{attribute 'GeneratedUsingTerminal: EK1100-0000-0018'}
{attribute addProperty BoxType "EK1100-0000-0018"}
{attribute addProperty Id "Beckhoff_EJ3xxxEK1122Beckhoff_EJ3xxxEK1122_F46733132A_0001_EJ3004_0000_0019EJ3004_9DDA7BAE48A_0002_EJ3004_0000_0020EJ3004_9DDA7BAE48A_0003_EJ3004_0000_0021EJ3004_9DDA7BAE48A_0004_EJ3048_0000_0020EJ3048_085DE50284A_0005_EJ3058_0000_0020EJ3058_085DE50284A_0006_EJ3068_0000_0020EJ3068_085DE50284A_0007_EJ3068_0000_0021EJ3068_085DE50284A_0008_EJ3104_0000_0019EJ3104_0E4717A052A_0009_EJ3104_0000_0020EJ3104_0E4717A052A_0010_EJ3104_0000_0021EJ3104_0E4717A052A_0011_EJ3108_0000_0017EJ3108_085DE50284A_0012_EJ3108_0000_0018EJ3108_5798389192A_0013_EJ3108_0000_0019EJ3108_5798389192A_0014_EJ3202_0000_0019EJ3202_14BDD8A530A_0015_EJ3202_0000_0020EJ3202_14BDD8A530A_0016_EJ3202_0000_0021EJ3202_14BDD8A530A_0017_EJ3214_0000_0016EJ3214_AFE9644F40A_0018_EJ3255_0000_0023EJ3255_6B0AD73762A_0019_EJ3318_0000_0017EJ3318_CF36AC5082"}
{attribute addProperty CRC "449149787"}
{attribute addProperty Size "1180"}
TYPE Beckhoff_EJ3xxx_1AC57B5B EXTENDS EK1100_AB5A9467 :
STRUCT
	{attribute addProperty Name "Beckhoff_EJ3xxxEK1122"}
	{attribute addProperty PreviousPort "Beckhoff EJ3xxx : B"}
	Beckhoff_EJ3xxxEK1122 : Beckhoff_EJ3xxxEK1122_F4673313;
	{attribute addProperty Name "A_0001_EJ3004_0000_0019"}
	{attribute addProperty PreviousPort "Beckhoff EJ3xxxEK1122 : C"}
	A_0001_EJ3004_0000_0019 : EJ3004_9DDA7BAE;
	{attribute addProperty Name "A_0002_EJ3004_0000_0020"}
	{attribute addProperty PreviousPort "A_0001(EJ3004-0000-0019) : B"}
	A_0002_EJ3004_0000_0020 : EJ3004_9DDA7BAE;
	{attribute addProperty Name "A_0003_EJ3004_0000_0021"}
	{attribute addProperty PreviousPort "A_0002(EJ3004-0000-0020) : B"}
	A_0003_EJ3004_0000_0021 : EJ3004_9DDA7BAE;
	{attribute addProperty Name "A_0004_EJ3048_0000_0020"}
	{attribute addProperty PreviousPort "A_0003(EJ3004-0000-0021) : B"}
	A_0004_EJ3048_0000_0020 : EJ3048_085DE502;
	{attribute addProperty Name "A_0005_EJ3058_0000_0020"}
	{attribute addProperty PreviousPort "A_0004(EJ3048-0000-0020) : B"}
	A_0005_EJ3058_0000_0020 : EJ3058_085DE502;
	{attribute addProperty Name "A_0006_EJ3068_0000_0020"}
	{attribute addProperty PreviousPort "A_0005(EJ3058-0000-0020) : B"}
	A_0006_EJ3068_0000_0020 : EJ3068_085DE502;
	{attribute addProperty Name "A_0007_EJ3068_0000_0021"}
	{attribute addProperty PreviousPort "A_0006(EJ3068-0000-0020) : B"}
	A_0007_EJ3068_0000_0021 : EJ3068_085DE502;
	{attribute addProperty Name "A_0008_EJ3104_0000_0019"}
	{attribute addProperty PreviousPort "A_0007(EJ3068-0000-0021) : B"}
	A_0008_EJ3104_0000_0019 : EJ3104_0E4717A0;
	{attribute addProperty Name "A_0009_EJ3104_0000_0020"}
	{attribute addProperty PreviousPort "A_0008(EJ3104-0000-0019) : B"}
	A_0009_EJ3104_0000_0020 : EJ3104_0E4717A0;
	{attribute addProperty Name "A_0010_EJ3104_0000_0021"}
	{attribute addProperty PreviousPort "A_0009(EJ3104-0000-0020) : B"}
	A_0010_EJ3104_0000_0021 : EJ3104_0E4717A0;
	{attribute addProperty Name "A_0011_EJ3108_0000_0017"}
	{attribute addProperty PreviousPort "A_0010(EJ3104-0000-0021) : B"}
	A_0011_EJ3108_0000_0017 : EJ3108_085DE502;
	{attribute addProperty Name "A_0012_EJ3108_0000_0018"}
	{attribute addProperty PreviousPort "A_0011(EJ3108-0000-0017) : B"}
	A_0012_EJ3108_0000_0018 : EJ3108_57983891;
	{attribute addProperty Name "A_0013_EJ3108_0000_0019"}
	{attribute addProperty PreviousPort "A_0012(EJ3108-0000-0018) : B"}
	A_0013_EJ3108_0000_0019 : EJ3108_57983891;
	{attribute addProperty Name "A_0014_EJ3202_0000_0019"}
	{attribute addProperty PreviousPort "A_0013(EJ3108-0000-0019) : B"}
	A_0014_EJ3202_0000_0019 : EJ3202_14BDD8A5;
	{attribute addProperty Name "A_0015_EJ3202_0000_0020"}
	{attribute addProperty PreviousPort "A_0014(EJ3202-0000-0019) : B"}
	A_0015_EJ3202_0000_0020 : EJ3202_14BDD8A5;
	{attribute addProperty Name "A_0016_EJ3202_0000_0021"}
	{attribute addProperty PreviousPort "A_0015(EJ3202-0000-0020) : B"}
	A_0016_EJ3202_0000_0021 : EJ3202_14BDD8A5;
	{attribute addProperty Name "A_0017_EJ3214_0000_0016"}
	{attribute addProperty PreviousPort "A_0016(EJ3202-0000-0021) : B"}
	A_0017_EJ3214_0000_0016 : EJ3214_AFE9644F;
	{attribute addProperty Name "A_0018_EJ3255_0000_0023"}
	{attribute addProperty PreviousPort "A_0017(EJ3214-0000-0016) : B"}
	A_0018_EJ3255_0000_0023 : EJ3255_6B0AD737;
	{attribute addProperty Name "A_0019_EJ3318_0000_0017"}
	{attribute addProperty PreviousPort "A_0018(EJ3255-0000-0023) : B"}
	A_0019_EJ3318_0000_0017 : EJ3318_CF36AC50;
END_STRUCT
END_TYPE

(* stored: Version 1.2.0.0, ProductVersion 3.1.4024.9
   DUT Beckhoff_EJ3xxx_1AC57B5B: Id {8e3115a0-ea6f-4c19-b2e1-2a5091041487} *)
